// Mitsubishi GX Works2 project: 인버터 컨베어   PLC: Q03UDV

PROGRAM MAIN
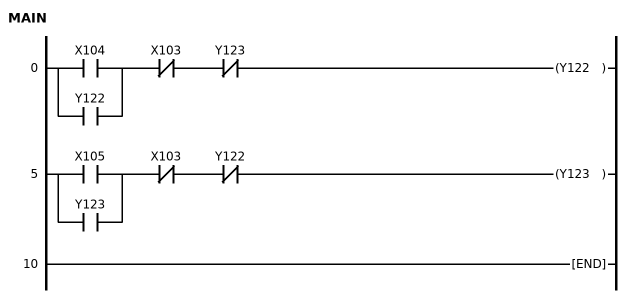
0     LD      X104
      OR      Y122
      ANI     X103
      ANI     Y123
      OUT     Y122
5     LD      X105
      OR      Y123
      ANI     X103
      ANI     Y122
      OUT     Y123
10    END
END_PROGRAM
